Fanuc KAREL source: tst_csv_rdln.kl

PROGRAM tst_csv_rdln
%NOLOCKGROUP

CONST
  CSV_NAME = 'FR:\read_data.csv'
  SAMPLE_TIME = 100

VAR
  fl : FILE
  pose : XYZWPR
  header : STRING[12]
  str : STRING[64]
  b : BOOLEAN

%include display.c.klt
%include systemlib.codes.klt
%include systemlib.datatypes.klt

%from display.klh %import clear, show
%from strings.klh %import pose_to_s, s_to_xyzwpr
%include csv.klh

BEGIN
  --open csv file
  csv__read_open(CSV_NAME, fl)
  --read header
  header = csv__read_line(CSV_NAME, fl)

  --clear display
  display__clear
  --show display
  display__show
  WRITE TPDISPLAY(CR,CR)

  REPEAT
    b = csv__read_line_ref(CSV_NAME, fl, str)
    IF b THEN
      pose = s_to_xyzwpr(str, ',')

      WRITE TPDISPLAY(pose_to_s(pose,','),CR)
    ENDIF

    DELAY SAMPLE_TIME
  UNTIL(NOT b)

  csv__read_close(fl)

  WRITE TPDISPLAY('Read finished!',CR)

END tst_csv_rdln
